// Mitsubishi GX Works2 project: LRI.gx3_SEMÁFARO 01   PLC: Q03UDV

FUNCTION_BLOCK BLOCK1
VAR_INPUT
  Start : BOOL;
  OFFStop : BOOL;
END_VAR
VAR_OUTPUT
  Relay : BOOL;
END_VAR
VAR
  Timer0 : TIMER;
  Timer2 : TIMER;
  Timer1 : TIMER;
END_VAR
VAR_OUTPUT
  Lamp1 : BOOL;
  Lamp2 : BOOL;
END_VAR
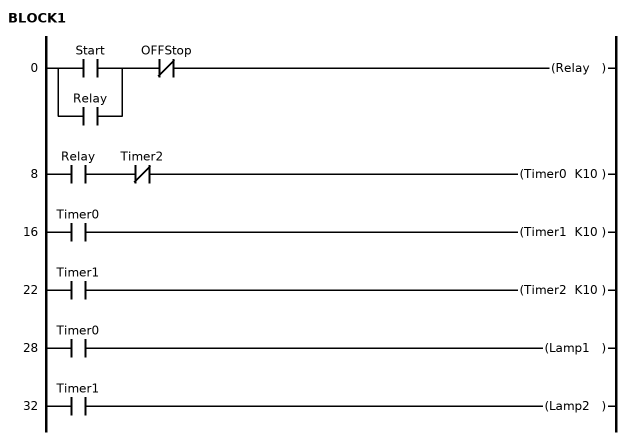
0     LD      Start
      OR      Relay
      ANI     OFFStop
      OUT     Relay
8     LD      Relay
      ANI     Timer2
      OUT     Timer0 K10
16    LD      Timer0
      OUT     Timer1 K10
22    LD      Timer1
      OUT     Timer2 K10
28    LD      Timer0
      OUT     Lamp1
32    LD      Timer1
      OUT     Lamp2
END_FUNCTION_BLOCK

PROGRAM Monitor
VAR
  BLOCK1_1 : BLOCK1;
  BLOCK1_2 : BLOCK1;
  BLOCK1_3 : BLOCK1;
  BLOCK1_4 : BLOCK1;
END_VAR
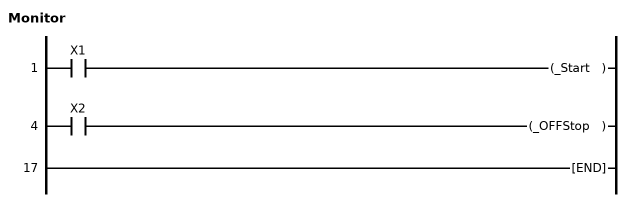
; FB BLK START BLOCK1(BLOCK1_4)
1     LD      X1
      OUT     _Start
4     LD      X2
      OUT     _OFFStop
; FB START
; FB_NAME BLOCK1
; INSTANCE_NAME BLOCK1_4
; FB IN_B:Start
; FB OUT_Relay:B
; FB IN_B:OFFStop
; FB OUT_Lamp1:B
; FB OUT_Lamp2:B
; FB END
; FB BLK END
17    END
END_PROGRAM
